// TIA Portal V15 export
// export: Created 2019-01-03T10:58:21.1379348Z, ExportSetting WithDefaults, WithReadOnly, DisplayName Totally Integrated Automation Portal, DisplayVersion V15 Update 2, DisplayName TIA Portal Openness, DisplayVersion V15 Update 2, DisplayName STEP 7 Professional, DisplayVersion V15 Update 2, DisplayName STEP 7 Safety, DisplayVersion V15, DisplayName WinCC Professional, DisplayVersion V15 Update 2, DisplayName SIMATIC Visualization Architect, DisplayVersion V15 Update 1
DATA_BLOCK "FGDB_040XSK001"   // DB158
TITLE = 040GST001 sequence / 040GST001 Ablaufkette
{ S7_Optimized_Access := 'FALSE' }
AUTHOR : integra
FAMILY : GF
VERSION : 0.1
// stored: AutoNumber true, CodeModifiedDate 2018-01-29T16:41:46.858993Z, CompileDate 2018-02-20T10:24:47.6269504Z, CreationDate 2017-05-30T07:46:55.5707793Z, DBAccessibleFromOPCUA true, InstanceOfName iFG_GRAPH_CONTROL, InstanceOfNumber 1014, InstanceOfType FB, InterfaceModifiedDate 2018-01-24T12:13:15.0981281Z, IsConsistent true, IsKnowHowProtected false, ModifiedDate 2018-01-29T16:41:46.858993Z, ParameterModified 2017-05-11T15:58:30.7257784Z, StructureModified 2017-06-01T12:07:06.3112253Z, UDAEnableTagReadback false
"iFG_GRAPH_CONTROL"
   // VAR_INPUT
   //    fct : Int;
   //    safetyStop : Bool;
   //    enableOut : Bool;
   //    actionOff : Bool;
   //    jog : Bool;
   //    jogPlus_1 : Bool;
   //    init : Bool;
   //    haltStepN : Bool;
   // END_VAR
   // VAR_OUTPUT
   //    fault : Bool;
   //    faultExt : Bool;
   // END_VAR
   // VAR_IN_OUT
   //    GRAPH_Extension : "iUDT_GRAPH_EXTENSION";
   // END_VAR
   // VAR RETAIN
   //    idx : Int;
   //    sectionNumber : Int;
   //    deskNumber : Int;
   //    stationNumber : Int;
   //    dbNumber : Int;
   //    function : Int;
   //    numberInternalMessages : Int;
   //    numberExternalMessages : Int;
   //    Settings : Struct
   //       haltStepN { S7_SetPoint := 'True'} : Int;
   //       stepNumber { S7_SetPoint := 'True'} : Int;
   //       immediatelyFault { S7_SetPoint := 'True'} : Bool;
   //    END_STRUCT;
   //    F : Struct
   //       fct : Bool;
   //       sequenceFault : Bool;
   //       immediatelyFault : Bool;
   //       versionConflict : Bool;
   //       stepNotExist : Bool;
   //    END_STRUCT;
   //    "M" : Struct
   //       more_1_sequence : Bool;
   //       more_16_simultanBranch : Bool;
   //       more_16_transition : Bool;
   //    END_STRUCT;
   //    Masks : Struct
   //       disableFault_1_8 : Byte;
   //       prodRelevantFault_1_8 : Byte;
   //    END_STRUCT;
   //    LastState : Struct
   //       fault_1_8 : Byte;
   //       message_1_8 : Byte;
   //    END_STRUCT;
   //    IfcFGExternal : "iUDT_IFC_SYS_EXTERNAL_ALARM";
   //    Tmr : Struct
   //       s_1 { S7_SetPoint := 'True'} : Int;
   //       s_2 { S7_SetPoint := 'True'} : Int;
   //    END_STRUCT;
   //    ExtP : Struct
   //       setup : Bool;
   //       auto : Bool;
   //       enableIn : Bool;
   //       ack : Bool;
   //    END_STRUCT;
   //    StM : Struct
   //       fault : Bool;
   //       setup : Bool;
   //       auto : Bool;
   //       warning : Bool;
   //       eStop : Bool;
   //       safetyStop : Bool;
   //       enableIn : Bool;
   //       enableOutForward : Bool;
   //       enableOutBackward : Bool;
   //       faultPr : Bool;
   //       pairMon : Bool;
   //       specialMode : Bool;
   //       "13" : Bool;
   //       "14" : Bool;
   //       "15" : Bool;
   //       "16" : Bool;
   //       "17" : Bool;
   //       "18" : Bool;
   //       "19" : Bool;
   //       "20" : Bool;
   //       "21" : Bool;
   //       "22" : Bool;
   //       "23" : Bool;
   //       "24" : Bool;
   //       "25" : Bool;
   //       "26" : Bool;
   //       "27" : Bool;
   //       "28" : Bool;
   //       "29" : Bool;
   //       "30" : Bool;
   //       "31" : Bool;
   //       "32" : Bool;
   //    END_STRUCT;
   //    VB : Struct
   //       init : Bool;
   //       toStepN : Bool;
   //       inStepN : Bool;
   //       "4" : Bool;
   //       "5" : Bool;
   //       "6" : Bool;
   //       "7" : Bool;
   //       "8" : Bool;
   //       "9" : Bool;
   //       "10" : Bool;
   //       "11" : Bool;
   //       "12" : Bool;
   //       "13" : Bool;
   //       "14" : Bool;
   //       "15" : Bool;
   //       "16" : Bool;
   //       "17" : Bool;
   //       "18" : Bool;
   //       "19" : Bool;
   //       "20" : Bool;
   //       "21" : Bool;
   //       "22" : Bool;
   //       "23" : Bool;
   //       "24" : Bool;
   //       "25" : Bool;
   //       "26" : Bool;
   //       "27" : Bool;
   //       "28" : Bool;
   //       "29" : Bool;
   //       "30" : Bool;
   //       "31" : Bool;
   //       "32" : Bool;
   //    END_STRUCT;
   //    VCB : Struct
   //       ack : Bool;
   //       init : Bool;
   //       smartSync : Bool;
   //    END_STRUCT;
   //    D : Struct
   //       immediatelyFault : Bool;
   //       visuAck : Bool;
   //       enableIn : Bool;
   //       visuInit : Bool;
   //       init : Bool;
   //       fPInit : Bool;
   //       pPInit : Bool;
   //       pPToInit : Bool;
   //       fPToInit : Bool;
   //       auto : Bool;
   //       fNAuto : Bool;
   //       pNAuto : Bool;
   //       fPAuto : Bool;
   //       pPAuto : Bool;
   //       fNSpecial : Bool;
   //       pNSpecial : Bool;
   //       fPSpecial : Bool;
   //       pPSpecial : Bool;
   //       specialPlus_1 : Bool;
   //       fPSpecialPlus_1 : Bool;
   //       pPSpecialPlus_1 : Bool;
   //       fPHaltStepN : Bool;
   //       pPHaltStepN : Bool;
   //       fPStepError : Bool;
   //       fPStepNotExist : Bool;
   //       haltStepNActive : Bool;
   //       haltStepNReady : Bool;
   //       startSmartSync : Bool;
   //    END_STRUCT;
   //    V : Struct
   //       runtime : UInt;
   //    END_STRUCT;
   //    GRAPH : "iUDT_GRAPH_EXTENSION";
   // END_VAR
BEGIN
END_DATA_BLOCK
